// Valid on Done (S3.12).
TYPE ST_AxisOutCmd :
STRUCT
    InPosition : BOOL;
    Homed      : BOOL;
END_STRUCT
END_TYPE

(* stored: Version 1.1.0.1, ProductVersion 3.1.4024.12
   DUT ST_AxisOutCmd: Id {965932d8-8353-44d8-b0e1-9c0a50b76513} *)
